{attribute 'pack_mode' := '1'}
TYPE ST_ReadVehicleData :
STRUCT
	stReadListReturnInfo		: ARRAY [1..1] OF ST_UAReadListReturnInfo;
	stVehicle					: ST_StatusVehicle;

END_STRUCT
END_TYPE

(* stored: Version 1.1.0.1, ProductVersion 3.1.4024.5
   DUT ST_ReadVehicleData: Id {02046c2c-17a5-4365-9af3-5b6848f1e244} *)
